Fanuc KAREL source: kt00745.KL

-- PROVISIONAL review KL for V770-1; original PC SHA256 09f142e57bf0b3e324960f5ce9283a6cbafe9e2158f956b30da0d15d84b9186e
-- Incomplete behavior may be omitted. Consult companion uncertainty JSON. Do not deploy.
PROGRAM KT00745
%NOLOCKGROUP
BEGIN
  -- UNRESOLVED_PC offsets 5-18; opcodes 22,1D,23
  -- UNRESOLVED_PC offsets 23-27; opcodes 7F
END KT00745
